TYPE defItem :
STRUCT
	Counter AT%I* : BYTE;
	Bound AT%Q* : BYTE;
	PitchX AT%Q* : REAL;
	PitchY AT%Q* : REAL;
END_STRUCT
END_TYPE

(* stored: Version 1.1.0.1, ProductVersion 3.1.4024.0
   DUT defItem: Id {40371373-15e9-464c-9148-8d025db7018a} *)
